{attribute 'qualified_only'}
VAR_GLOBAL CONSTANT
	LOG_FOLDER : STRING := ''; // Location for the log files
END_VAR

(* stored: Version 1.1.0.1, ProductVersion 3.1.4024.11
   GVL PAR_System: Id {5a55aa4b-3439-04ae-03bc-3258d3bc63e5}, ParameterList True *)
